TEXTLIST TextList_Canne_Transfert
  0 = 'Canne\t' | FR: 'Canne de transfert' | EN: 'Transfer arm'
  1 = 'Position' | FR: 'Position' | EN: 'Position'
  2 = 'Speed' | FR: 'Vitesse' | EN: 'Speed'
  3 = 'Poste' | FR: 'Position correspondante' | EN: 'Corresponding position'
  4 = 'Poste choisi' | FR: 'Position sélectionnée' | EN: 'Selected position'
  5 = 'Distance' | FR: 'Distance' | EN: 'Distance'
  6 = 'vitesse' | FR: 'Vitesse' | EN: 'Speed'
  7 = 'controle' | FR: 'Opération' | EN: 'Operation'
  8 = 'Durée' | FR: 'Durée : ' | EN: 'Duration:'
  9 = 'ecoulée' | FR: 'Durée écoulée :' | EN: 'Elapsed time:'
   = ''
END_TEXTLIST

(* stored: Version 1.1.0.1, ProductVersion 3.1.4024.10
   TextList TextList_Canne_Transfert: Id {0c11cbd1-66e4-4dec-bac1-2e1fcad1e4dd} *)
